// TIA Portal V19 export
DATA_BLOCK "DB_CurrentRecipe"   // DB5
{ S7_Optimized_Access := 'TRUE'; DB_Accessible_From_OPC_UA := 'FALSE' }
// stored: AutoNumber false, DBAccessibleFromOPCUA false, DBAccessibleFromWebserver false, MemoryReserve 100
   VAR RETAIN
      usiCurrentRecipeNumber : USInt;
      usiCurrentLayerType : USInt;
      usiCurrentJobDataLeft { ExternalAccessible := 'False'; ExternalVisible := 'False'; ExternalWritable := 'False'} : USInt;
      usiCurrentJobDataRight { ExternalAccessible := 'False'; ExternalVisible := 'False'; ExternalWritable := 'False'} : USInt;
      uiCdbNumber : UInt;
      CompleteRecipe : "stRecipe";
      WorkRecipe { S7_SetPoint := 'True'} : "stWorkRecipe";
   END_VAR
BEGIN
END_DATA_BLOCK
